FUNCTION P2CHAR : CHAR
VAR_INPUT
	p : POINTER TO STRING;
END_VAR
VAR
END_VAR

P2CHAR := p^;

END_FUNCTION

(* stored: Version 1.1.0.1, ProductVersion 3.1.4024.11
   POU P2CHAR: Id {4a6f9bdc-5292-46ed-9071-7292be1a6e29}, SpecialFunc None *)
